PROGRAM MAIN
VAR
	Loadcells			: FB_Loadcells(ModbusAddresses:= LoadcellAddresses, ReadPeriod:= T#1s);
	LoadsInKg			: ARRAY[1..MAX_LOADCELLS] OF INT; //loads on loadcells
END_VAR
VAR CONSTANT
	MAX_LOADCELLS		: UINT:= 10;
	LoadcellAddresses	: ARRAY[1..MAX_LOADCELLS] OF BYTE:= [1,2,3,4,0]; //must end with 0
END_VAR

Loadcells.Cyclic(LoadsInKg:= LoadsInKg);

END_PROGRAM

(* stored: Version 1.1.0.1, ProductVersion 3.1.4024.15
   POU MAIN: Id {68d2e4c8-fc37-4655-8c1a-780d28187236}, SpecialFunc None *)
